# EPICS autosave request: support/ip/2-9/ipApp/Db/Pelco_CM6700_settings.req
$(P)$(R)Mon1.VAL
$(P)$(R)Mon2.VAL
$(P)$(R)Mon3.VAL
$(P)$(R)Mon4.VAL
$(P)$(R)Mon1.DESC
$(P)$(R)Mon2.DESC
$(P)$(R)Mon3.DESC
$(P)$(R)Mon4.DESC
$(P)$(R)Mon1.ZRST
$(P)$(R)Mon1.ONST
$(P)$(R)Mon1.TWST
$(P)$(R)Mon1.THST
$(P)$(R)Mon1.FRST
$(P)$(R)Mon1.FVST
$(P)$(R)Mon1.SXST
$(P)$(R)Mon1.SVST
$(P)$(R)Mon1.EIST
$(P)$(R)Mon1.NIST
$(P)$(R)Mon1.TEST
$(P)$(R)Mon1.ELST
$(P)$(R)Mon1.TVST
$(P)$(R)Mon1.TTST
$(P)$(R)Mon1.FTST
$(P)$(R)Mon1.FFST
